PROGRAM MAIN
VAR
END_VAR

END_PROGRAM

(* stored: Version 1.1.0.1
   POU MAIN: Id {5d158e57-baec-4634-a25e-b5e14c574c3e} *)
